FUNCTION_BLOCK Room_Ctx_Priv
VAR_INPUT
	bReady		: BOOL;
	bOpen		: BOOL;
	bClosed		: BOOL;
	bPaused		: BOOL;
	bAbort		: BOOL;
END_VAR

END_FUNCTION_BLOCK

(* stored: Version 1.1.0.1
   POU Room_Ctx_Priv: Id {f780ea0b-40f4-4a65-aec6-edfe7e6fb652}, SpecialFunc None *)
